FUNCTION_BLOCK Kommunikation
VAR_INPUT
END_VAR
VAR_OUTPUT
END_VAR
VAR
END_VAR

END_FUNCTION_BLOCK

(* stored: Version 1.1.0.1, ProductVersion 3.1.4024.13
   POU Kommunikation: Id {819753f2-3217-43d9-848a-d77cf7327dce}, SpecialFunc None *)
